FUNCTION_BLOCK ODriveAxisController
VAR_INPUT
	NodeId : UINT;
END_VAR

VAR_OUTPUT
	
END_VAR

VAR
	_fbODriveCanSimpleTransporter : ODriveCanSimpleTransporter;
END_VAR

_fbODriveCanSimpleTransporter();

METHOD GetError
VAR_INPUT
	bExecute : BOOL;
END_VAR

VAR_OUTPUT
	bBusy : BOOL;
	bError : BOOL;
	sErrorMsg : STRING;
	bDone : BOOL;
	stOdriveError : ST_OdriveError;
END_VAR

VAR
	stCanMsg : ST_CanMessage;
	nRTR : UINT := 1;
	
	bAddCmdDone : BOOL;
	bDataExist : BOOL;
	
	nIdx : UINT;
END_VAR

VAR_INST
	nStep : UINT;
	rTrig : R_TRIG;
	tmrTimeOut : TON;
	uOdriveError : U_OdriveErrorBytes;
END_VAR
CASE nStep OF
	0:	// Idle
		rTrig(CLK:= bExecute);
		IF rTrig.Q THEN
			bBusy := TRUE;			
			nStep := 1;
		END_IF
	
	1: // Add command
		stCanMsg.CobId := SHL(SHL(NodeId, 5) OR TO_UINT(E_OdriveCmd.GetError), 5) OR SHL(nRTR, 4);
		_fbODriveCanSimpleTransporter.AddCmd(stCanMsg, bDone=> bAddCmdDone, bError=> bError, sErrorMsg=> sErrorMsg);
		IF bAddCmdDone THEN
			bBusy := TRUE;
			nStep := 2;
		END_IF
		
	2: // Receive command
		_fbODriveCanSimpleTransporter.ReceiveData(NodeId, E_OdriveCmd.GetError, bExist=> bDataExist, stResultCanMsg=> stCanMsg);
		tmrTimeOut(IN:= TRUE, PT:= GVL_ODrive.nReceiveData_TimeOut);
		
		IF tmrTimeOut.Q THEN	// Time out
			bError := TRUE;
			sErrorMsg := 'Time out !';
			
		ELSIF NOT bDataExist THEN	// Not receive data yet
			bBusy := TRUE;
			
		ELSE	// Receive data
			bDone := TRUE;
			FOR nIdx := 0 TO 7 DO
				uOdriveError.aBytes[nIdx] := stCanMsg.Data[nIdx];
			END_FOR
			stOdriveError := uOdriveError.stOdriveError;
			nStep := 3;
		END_IF
	
	3:	// Finish
		IF bExecute THEN
			bDone := TRUE;
			stOdriveError := uOdriveError.stOdriveError;
			
		ELSE
			bDone := FALSE;
			rTrig(CLK:= FALSE);
			tmrTimeOut(IN:= FALSE);
			nStep := 0;
		END_IF
	
END_CASE
END_METHOD

METHOD GetEncoderEstimates
VAR_INPUT
	bExecute : BOOL;
END_VAR

VAR_OUTPUT
	bBusy : BOOL;
	bError : BOOL;
	sErrorMsg : STRING;
	bDone : BOOL;
	stOdriveEncoderEstimates : ST_OdriveEncoderEstimates;
END_VAR

VAR
	stCanMsg : ST_CanMessage;
	nRTR : UINT := 1;
	
	bAddCmdDone : BOOL;
	bDataExist : BOOL;
	
	nIdx : UINT;
END_VAR

VAR_INST
	nStep : UINT;
	rTrig : R_TRIG;
	tmrTimeOut : TON;
	uEncoderEstimates : U_OdriveEncoderEstimatesBytes;
END_VAR
CASE nStep OF
	0:	// Idle
		rTrig(CLK:= bExecute);
		IF rTrig.Q THEN
			bBusy := TRUE;			
			nStep := 1;
		END_IF
	
	1: // Add command
		stCanMsg.CobId := SHL(SHL(NodeId, 5) OR TO_UINT(E_OdriveCmd.GetEncoderEstimates), 5) OR SHL(nRTR, 4);
		_fbODriveCanSimpleTransporter.AddCmd(stCanMsg, bDone=> bAddCmdDone, bError=> bError, sErrorMsg=> sErrorMsg);
		IF bAddCmdDone THEN
			bBusy := TRUE;
			nStep := 2;
		END_IF
		
	2: // Receive command
		_fbODriveCanSimpleTransporter.ReceiveData(NodeId, E_OdriveCmd.GetEncoderEstimates, bExist=> bDataExist, stResultCanMsg=> stCanMsg);
		tmrTimeOut(IN:= TRUE, PT:= GVL_ODrive.nReceiveData_TimeOut);
		
		IF tmrTimeOut.Q THEN	// Time out
			bError := TRUE;
			sErrorMsg := 'Time out !';
			
		ELSIF NOT bDataExist THEN	// Not receive data yet
			bBusy := TRUE;
			
		ELSE	// Receive data
			bDone := TRUE;
			FOR nIdx := 0 TO 7 DO
				uEncoderEstimates.aBytes[nIdx] := stCanMsg.Data[nIdx];
			END_FOR
			stOdriveEncoderEstimates := uEncoderEstimates.stEncoderEstimates;
			nStep := 3;
		END_IF
	
	3:	// Finish
		IF bExecute THEN
			bDone := TRUE;
			stOdriveEncoderEstimates := uEncoderEstimates.stEncoderEstimates;
			
		ELSE
			bDone := FALSE;
			rTrig(CLK:= FALSE);
			tmrTimeOut(IN:= FALSE);
			nStep := 0;
		END_IF
	
END_CASE
END_METHOD

METHOD GetHeartBeat
VAR_INPUT
	bExecute : BOOL;
END_VAR

VAR_OUTPUT
	bBusy : BOOL;
	bError : BOOL;
	sErrorMsg : STRING;
	bDone : BOOL;
	stOdriveHeartBeat : ST_OdriveHeartbeat;
END_VAR

VAR
	stCanMsg : ST_CanMessage;
	nRTR : UINT := 1;
	
	bAddCmdDone : BOOL;
	bDataExist : BOOL;
	
	nIdx : UINT;
END_VAR

VAR_INST
	nStep : UINT;
	rTrig : R_TRIG;
	tmrTimeOut : TON;
	uOdriveHeartBeat : U_OdriveHeartbeatBytes;
END_VAR
CASE nStep OF
	0:	// Idle
		rTrig(CLK:= bExecute);
		IF rTrig.Q THEN
			bBusy := TRUE;			
			nStep := 1;
		END_IF
	
	1: // Add command
		stCanMsg.CobId := SHL(SHL(NodeId, 5) OR TO_UINT(E_OdriveCmd.Heartbeat), 5) OR SHL(nRTR, 4);
		_fbODriveCanSimpleTransporter.AddCmd(stCanMsg, bDone=> bAddCmdDone, bError=> bError, sErrorMsg=> sErrorMsg);
		IF bAddCmdDone THEN
			bBusy := TRUE;
			nStep := 2;
		END_IF
		
	2: // Receive command
		_fbODriveCanSimpleTransporter.ReceiveData(NodeId, E_OdriveCmd.Heartbeat, bExist=> bDataExist, stResultCanMsg=> stCanMsg);
		tmrTimeOut(IN:= TRUE, PT:= GVL_ODrive.nReceiveData_TimeOut);
		
		IF tmrTimeOut.Q THEN	// Time out
			bError := TRUE;
			sErrorMsg := 'Time out !';
			
		ELSIF NOT bDataExist THEN	// Not receive data yet
			bBusy := TRUE;
			
		ELSE	// Receive data
			bDone := TRUE;
			FOR nIdx := 0 TO 6 DO
				uOdriveHeartBeat.aBytes[nIdx] := stCanMsg.Data[nIdx];
			END_FOR
			stOdriveHeartBeat := uOdriveHeartBeat.stHeartbeat;
			nStep := 3;
		END_IF
	
	3:	// Finish
		IF bExecute THEN
			bDone := TRUE;
			stOdriveHeartBeat := uOdriveHeartBeat.stHeartbeat;
			
		ELSE
			bDone := FALSE;
			rTrig(CLK:= FALSE);
			tmrTimeOut(IN:= FALSE);
			nStep := 0;
		END_IF
	
END_CASE
END_METHOD

END_FUNCTION_BLOCK

(* stored: Version 1.1.0.1
   POU ODriveAxisController: Id {888f14a2-28b4-442c-8d2b-90ee242187e2}, SpecialFunc None
   Method GetError: Id {7ced9641-2f1e-4dcb-89a3-a01589153701}
   Method GetEncoderEstimates: Id {14a2520e-b7da-434d-8e95-8a742dcda8c6}
   Method GetHeartBeat: Id {cb9c0ea2-4e21-4d23-b1eb-ad5840aff9a5} *)
